// TIA Portal project "Automatic Coffee Machine" (V17)
// Automatic Coffee Machine
// The machine should dispense the appropriate amount of coffee for 5 seconds, then water for 10 seconds, followed by milk for 8 seconds. The process should end with a stirring of 5 seconds.

(* hardware
DEVICE "S7-1200 station_1"  S7-1200 Station
   slot 0: "Rack_0"  S7-1200 Rack  Rack  V1.0
   slot 1: "PLC_1"  CPU 1214C AC/DC/Rly  6ES7 214-1BG40-0XB0  V4.5
*)

// ===== PLC "PLC_1"  CPU 1214C AC/DC/Rly =====

VAR_GLOBAL   // PLC tag table "Default tag table"
   "Start button" AT %I0.0 : Bool;
   "Coffee dispenser" AT %Q0.0 : Bool;
   "Water valve/pump" AT %Q0.1 : Bool;
   "Milk dispenser" AT %Q0.2 : Bool;
   "Stirrer motor" AT %Q0.3 : Bool;
   "Tag_1" AT %M0.0 : Bool;
   "Tag_2" AT %M0.1 : Bool;
END_VAR

// folder: System blocks/Program resources

DATA_BLOCK "IEC_Timer_0_DB"   // DB1
{ S7_Optimized_Access := 'TRUE' }
AUTHOR : Simatic
FAMILY : IEC
NAME : IEC_TMR
VERSION : 1.0
// stored: InstanceOfName IEC_TIMER
"IEC_TIMER"
BEGIN
END_DATA_BLOCK

DATA_BLOCK "IEC_Timer_0_DB_1"   // DB2
{ S7_Optimized_Access := 'TRUE' }
AUTHOR : Simatic
FAMILY : IEC
NAME : IEC_TMR
VERSION : 1.0
// stored: InstanceOfName IEC_TIMER
"IEC_TIMER"
BEGIN
END_DATA_BLOCK

DATA_BLOCK "IEC_Timer_0_DB_2"   // DB3
{ S7_Optimized_Access := 'TRUE' }
AUTHOR : Simatic
FAMILY : IEC
NAME : IEC_TMR
VERSION : 1.0
// stored: InstanceOfName IEC_TIMER
"IEC_TIMER"
BEGIN
END_DATA_BLOCK

DATA_BLOCK "IEC_Timer_0_DB_3"   // DB4
{ S7_Optimized_Access := 'TRUE' }
AUTHOR : Simatic
FAMILY : IEC
NAME : IEC_TMR
VERSION : 1.0
// stored: InstanceOfName IEC_TIMER
"IEC_TIMER"
BEGIN
END_DATA_BLOCK

DATA_BLOCK "IEC_Timer_0_DB_4"   // DB5
{ S7_Optimized_Access := 'TRUE' }
AUTHOR : Simatic
FAMILY : IEC
NAME : IEC_TMR
VERSION : 1.0
// stored: InstanceOfName IEC_TIMER
"IEC_TIMER"
BEGIN
END_DATA_BLOCK

DATA_BLOCK "IEC_Timer_0_DB_5"   // DB6
{ S7_Optimized_Access := 'TRUE' }
AUTHOR : Simatic
FAMILY : IEC
NAME : IEC_TMR
VERSION : 1.0
// stored: InstanceOfName IEC_TIMER
"IEC_TIMER"
BEGIN
END_DATA_BLOCK

DATA_BLOCK "IEC_Timer_0_DB_6"   // DB7
{ S7_Optimized_Access := 'TRUE' }
AUTHOR : Simatic
FAMILY : IEC
NAME : IEC_TMR
VERSION : 1.0
// stored: InstanceOfName IEC_TIMER
"IEC_TIMER"
BEGIN
END_DATA_BLOCK

DATA_BLOCK "IEC_Timer_0_DB_7"   // DB8
{ S7_Optimized_Access := 'TRUE' }
AUTHOR : Simatic
FAMILY : IEC
NAME : IEC_TMR
VERSION : 1.0
// stored: InstanceOfName IEC_TIMER
"IEC_TIMER"
BEGIN
END_DATA_BLOCK

// folder: (top level)

ORGANIZATION_BLOCK "Main"   // OB1, LAD, ProgramCycle
TITLE = "Main Program Sweep (Cycle)"
{ S7_Optimized_Access := 'TRUE' }
VERSION : 0.1
   VAR_INPUT
      Initial_Call : Bool;   // Initial call of this OB
      Remanence : Bool;   // =True, if remanent data are available
   END_VAR
BEGIN

REGION Network 1
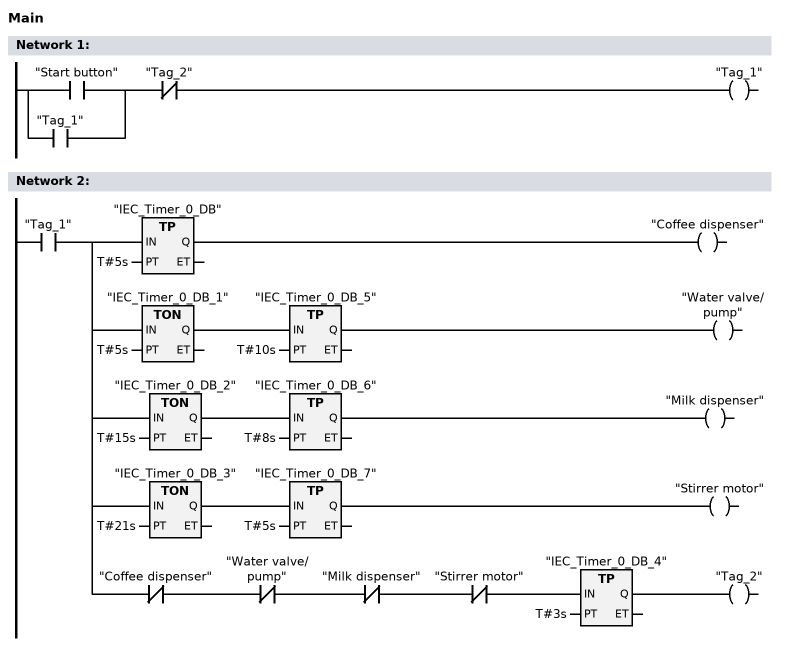
   RUNG wire#powerrail
      Contact( "Start button" )
      wire#w1
      I_Contact( "Tag_2" )
      Coil( "Tag_1" )
   END_RUNG
   RUNG wire#powerrail
      Contact( "Tag_1" )
   END_RUNG wire#w1
   // the same network as SCL:
   "Tag_1" := ("Start button" OR "Tag_1") AND NOT "Tag_2";
END_REGION

REGION Network 2
   "IEC_Timer_0_DB".TP(IN := "Tag_1", PT := T#5s);
   "Coffee dispenser" := "IEC_Timer_0_DB".Q;
   "IEC_Timer_0_DB_1".TON(IN := "Tag_1", PT := T#5s);
   "IEC_Timer_0_DB_5".TP(IN := "IEC_Timer_0_DB_1".Q, PT := T#10s);
   "Water valve/pump" := "IEC_Timer_0_DB_5".Q;
   "IEC_Timer_0_DB_2".TON(IN := "Tag_1", PT := T#15s);
   "IEC_Timer_0_DB_6".TP(IN := "IEC_Timer_0_DB_2".Q, PT := T#8s);
   "Milk dispenser" := "IEC_Timer_0_DB_6".Q;
   "IEC_Timer_0_DB_3".TON(IN := "Tag_1", PT := T#21s);
   "IEC_Timer_0_DB_7".TP(IN := "IEC_Timer_0_DB_3".Q, PT := T#5s);
   "Stirrer motor" := "IEC_Timer_0_DB_7".Q;
   "IEC_Timer_0_DB_4".TP(IN := "Tag_1" AND NOT "Coffee dispenser" AND NOT "Water valve/pump" AND NOT "Milk dispenser" AND NOT "Stirrer motor",
                         PT := T#3s);
   "Tag_2" := "IEC_Timer_0_DB_4".Q;
END_REGION
END_ORGANIZATION_BLOCK